FUNCTION_BLOCK FB_CloseOil
VAR_INPUT
END_VAR
VAR_OUTPUT
END_VAR
VAR
	idx			: INT;
END_VAR

FOR idx:=1 TO OilNo DO
	Oil[idx].IsOpen := FALSE;
	Oil[idx].CurTime := 0;
	Oil[idx].CloseStrokes := 0;
END_FOR

END_FUNCTION_BLOCK

(* stored: Version 1.1.0.1, ProductVersion 3.1.4024.9
   POU FB_CloseOil: Id {51976b35-578c-4822-84c0-982971712958}, SpecialFunc None *)
